FUNCTION F_TargetReached : BOOL
VAR_INPUT
	fCurrentPos: LREAL;
	fTargetPos: LREAL;
END_VAR


F_TargetReached := F_TargetWindowReached(fCurrentPos, fTargetPos, fEpsilon);

END_FUNCTION

(* stored: Version 1.1.0.1, ProductVersion 3.1.4022.9
   POU F_TargetReached: Id {b4785d9c-3817-4f5c-9628-573167cb6cb1}, SpecialFunc None *)
